// TwinCAT 3 PLC project TimersPractice
// ProgramVersion: 3.1.4024.0
// libraries:
//   Tc2_Standard, * (Beckhoff Automation GmbH)
//   Tc2_System, * (Beckhoff Automation GmbH)
//   Tc3_Module, * (Beckhoff Automation GmbH)
// project tree:
//   / PlcTask.TcTTO
//   POUs/ FB_TimerPulse.TcPOU, FB_Toggle.TcPOU, FB_Triggers.TcPOU, MAIN.TcPOU
// (motion and I/O tree: see PLC project instructions_practice)
// real-time tasks:
//   TASK PlcTask: cycle T#10ms, priority 20, ADS port 350
//   TASK PlcTask1: cycle T#10ms, priority 22, ADS port 351
//   TASK PlcTask2: cycle T#10ms, priority 21, ADS port 352
//   TASK PlcTask3: cycle T#10ms, priority 23, ADS port 353
//   TASK PlcTask4: cycle T#10ms, priority 24, ADS port 354
//   TASK PlcTask5: cycle T#10ms, priority 25, ADS port 355

CONFIGURATION TimersPractice
    RESOURCE PLC ON TwinCAT3
        TASK PlcTask(INTERVAL := T#10ms, PRIORITY := 24);
        PROGRAM MAIN WITH PlcTask : MAIN;
    END_RESOURCE
END_CONFIGURATION

// ---- POUs/MAIN.TcPOU
PROGRAM MAIN
VAR	
	fbToggle : FB_Toggle;
	fbTimerPulse : FB_TimerPulse;
	bStart : BOOL;
	fbTrigger : FB_Triggers;
END_VAR


IF bStart THEN
	fbTimerPulse();
	fbToggle();
	//fbTrigger();
END_IF

END_PROGRAM

// ---- POUs/FB_Toggle.TcPOU
FUNCTION_BLOCK FB_Toggle

VAR
	fbTon : TON := (PT := T#10S);
	bStart : BOOL := TRUE;
	fbTof : TOF := (PT := T#10S);
END_VAR

fbTon(IN := bStart);
IF fbTon.Q THEN
	bStart := FALSE;
END_IF
fbTof (IN := bStart);	
IF NOT fbTof.Q	THEN
	bStart := TRUE;
END_IF

END_FUNCTION_BLOCK

// ---- POUs/FB_TimerPulse.TcPOU
FUNCTION_BLOCK FB_TimerPulse

VAR
	fbTP : TP := (PT := T#10S);
	bResult : BOOL;
	bOn : BOOL;
END_VAR


fbTP(IN := bOn);
IF fbTP.Q THEN
	bResult := TRUE;
ELSE
	bResult  := FALSE;
END_IF

END_FUNCTION_BLOCK

// ---- POUs/FB_Triggers.TcPOU
FUNCTION_BLOCK FB_Triggers

VAR
	fbRTrig : R_TRIG;
	fbFTrig : F_TRIG;
	bTrigger : BOOL := TRUE;
	bRCount : INT ;
	bFCount : INT ;
	bCycleCount : UDINT ;
END_VAR

fbRTrig( CLK := bTrigger );
fbFTrig (CLK := bTrigger );
IF fbRTrig.Q THEN
	bRCount := bRCount + 1;
END_IF
IF fbFTrig.Q THEN
	bFCount := bFCount + 1;
END_IF
bCycleCount := bCycleCount + 1;

END_FUNCTION_BLOCK
